// TIA Portal V21 export
DATA_BLOCK "ADD_ON"   // DB263
{ S7_Optimized_Access := 'FALSE' }
   VAR RETAIN
      "SET TEMP1 STD3" : Real := 100.0;
      "SET TEMP2 STD3" : Real := 110.0;
      "SET TEMP3 STD3" : Real := 121.4;
      "SET PRESS STD3" : Real := 0.05;
      "SET HOLD1 STD3" : Int := 5;
      "SET HOLD2 STD3" : Int := 5;
      "SET HOLD3 STD3" : Int := 30;
      "SET VCC STD3" : Real := 0.0;
      "SET UP PRESS STD3" : Real := 0.0;
      "SET VCC HOLD STD3" : Int := 0;
      "SET NO OF PULSE STD3" : Int := 0;
      "SET TEMP1 STD4" : Real := 100.0;
      "SET TEMP2 STD4" : Real := 110.0;
      "SET TEMP3 STD4" : Real := 121.4;
      "SET PRESS STD4" : Real := 0.05;
      "SET HOLD1 STD4" : Int := 5;
      "SET HOLD2 STD4" : Int := 5;
      "SET HOLD3 STD4" : Int := 30;
      "SET VCC STD4" : Real := 0.0;
      "SET UP PRESS STD4" : Real := 0.0;
      "SET VCC HOLD STD4" : Int := 0;
      "SET NO OF PULSE STD4" : Int := 0;
      "SET TEMP1 STD5" : Real := 100.0;
      "SET TEMP2 STD5" : Real := 110.0;
      "SET TEMP3 STD5" : Real := 121.4;
      "SET PRESS STD5" : Real := 0.05;
      "SET HOLD1 STD5" : Int := 5;
      "SET HOLD2 STD5" : Int := 5;
      "SET HOLD3 STD5" : Int := 30;
      "SET VCC STD5" : Real := 0.0;
      "SET UP PRESS STD5" : Real := 0.0;
      "SET VCC HOLD STD5" : Int := 0;
      "SET NO OF PULSE STD5" : Int := 0;
      "SET TEMP1 STD6" : Real := 100.0;
      "SET TEMP2 STD6" : Real := 110.0;
      "SET TEMP3 STD6" : Real := 121.4;
      "SET PRESS STD6" : Real := 0.05;
      "SET HOLD1 STD6" : Int := 5;
      "SET HOLD2 STD6" : Int := 5;
      "SET HOLD3 STD6" : Int := 30;
      "SET VCC STD6" : Real := 0.0;
      "SET UP PRESS STD6" : Real := 0.0;
      "SET VCC HOLD STD6" : Int := 0;
      "SET NO OF PULSE STD6" : Int := 0;
      "SET TEMP1 STD7" : Real := 100.0;
      "SET TEMP2 STD7" : Real := 110.0;
      "SET TEMP3 STD7" : Real := 121.4;
      "SET PRESS STD7" : Real := 0.05;
      "SET HOLD1 STD7" : Int := 5;
      "SET HOLD2 STD7" : Int := 5;
      "SET HOLD3 STD7" : Int := 30;
      "SET VCC STD7" : Real := 0.0;
      "SET UP PRESS STD7" : Real := 0.0;
      "SET VCC HOLD STD7" : Int := 0;
      "SET NO OF PULSE STD7" : Int := 0;
      "SET TEMP1 STD8" : Real := 100.0;
      "SET TEMP2 STD8" : Real := 110.0;
      "SET TEMP3 STD8" : Real := 121.4;
      "SET PRESS STD8" : Real := 0.05;
      "SET HOLD1 STD8" : Int := 5;
      "SET HOLD2 STD8" : Int := 5;
      "SET HOLD3 STD8" : Int := 30;
      "SET VCC STD8" : Real := 0.0;
      "SET UP PRESS STD8" : Real := 0.0;
      "SET VCC HOLD STD8" : Int := 0;
      "SET NO OF PULSE STD8" : Int := 0;
      "SET TEMP1 STD9" : Real := 100.0;
      "SET TEMP2 STD9" : Real := 110.0;
      "SET TEMP3 STD9" : Real := 121.4;
      "SET PRESS STD9" : Real := 0.05;
      "SET HOLD1 STD9" : Int := 5;
      "SET HOLD2 STD9" : Int := 5;
      "SET HOLD3 STD9" : Int := 30;
      "SET VCC STD9" : Real := 0.0;
      "SET UP PRESS STD9" : Real := 0.0;
      "SET VCC HOLD STD9" : Int := 0;
      "SET NO OF PULSE STD9" : Int := 0;
      "SET LEAK VCC" : Real := -0.7;
      "SET VCC PRESS" : Real := -0.05;
      "SET DELAY BEFORE HOLD TIME" : Int := 0;
      "SET VCC HOLD TIME" : Int := 10;
      "SET ACCEPTANCE LEAK" : Real := 0.013;
   END_VAR
BEGIN
END_DATA_BLOCK
